TEXTLIST TextList_EnvironmentError
  0 = 'no_error'
  1 = 'not_connected'
  2 = 'invalid_state'
  3 = 'io_error'
  4 = 'unknown_error'
  666 = 'emergency_error'
   = ''
END_TEXTLIST

(* stored: Version 1.1.0.1, ProductVersion 3.1.4024.11
   TextList TextList_EnvironmentError: Id {a6669317-b045-4377-b00e-6b911d07e8dd} *)
